// TIA Portal V21 export
FUNCTION "chuj" : Void   // FC8, LAD
{ S7_Optimized_Access := 'TRUE' }
// stored: SetENOAutomatically false
BEGIN

REGION Network 1
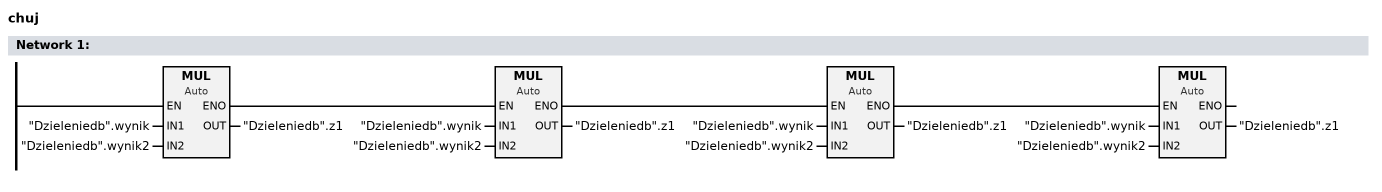
   RUNG wire#powerrail
      { S7_GenerateENO := "TRUE" } Mul(in1 := "Dzieleniedb".wynik, in2 := "Dzieleniedb".wynik2, out => "Dzieleniedb".z1)
      { S7_GenerateENO := "TRUE" } Mul(in1 := "Dzieleniedb".wynik, in2 := "Dzieleniedb".wynik2, out => "Dzieleniedb".z1)
      { S7_GenerateENO := "TRUE" } Mul(in1 := "Dzieleniedb".wynik, in2 := "Dzieleniedb".wynik2, out => "Dzieleniedb".z1)
      { S7_GenerateENO := "TRUE" } Mul(in1 := "Dzieleniedb".wynik, in2 := "Dzieleniedb".wynik2, out => "Dzieleniedb".z1)
   END_RUNG
   // the same network as SCL:
   // ENO of a box is taken as its EN; it also drops when the box reports an error
   "Dzieleniedb".z1 := "Dzieleniedb".wynik * "Dzieleniedb".wynik2;
   "Dzieleniedb".z1 := "Dzieleniedb".wynik * "Dzieleniedb".wynik2;
   "Dzieleniedb".z1 := "Dzieleniedb".wynik * "Dzieleniedb".wynik2;
   "Dzieleniedb".z1 := "Dzieleniedb".wynik * "Dzieleniedb".wynik2;
END_REGION
END_FUNCTION
